TYPE ST_ListMethod :
STRUCT
	methodName		: STRING(100);
	methodRevision	: STRING(100);
	
END_STRUCT
END_TYPE

(* stored: Version 1.1.0.1, ProductVersion 3.1.4024.15
   DUT ST_ListMethod: Id {9eaf245a-71d9-4657-8953-74f43bdc741a} *)
